{attribute 'qualified_only'}
{attribute 'strict'}
{attribute 'to_string'}
TYPE E_DruksensorStatus :
(
	SensorInputOk := 0,
	SensorInputError
);
END_TYPE

(* stored: Version 1.1.0.1
   DUT E_DruksensorStatus: Id {58ed60dd-09e9-41ae-a63b-2df7e7d4ed4b} *)
